{attribute 'linkalways'}
{attribute 'no_explicit_call' := 'This FB is a CLASS and must be accessed using methods or properties'}
{attribute 'enable_dynamic_creation'}
FUNCTION_BLOCK _ETcVnDetectBarcodesWalshOptions EXTENDS EnumDatatypeBase
VAR
	localData : ETcVnDetectBarcodesWalshOptions;
	activeData : REFERENCE TO ETcVnDetectBarcodesWalshOptions;
	enumBaseDatatype : _UDINT(localData);
END_VAR

METHOD PRIVATE AddLocalEnumeration
VAR_INPUT
	Enumeration : T_MAXSTRING;
	Value : ETcVnDetectBarcodesWalshOptions;
END_VAR
AddEnumeration(Enumeration, Value);
END_METHOD

PROPERTY PUBLIC Address : PVOID
GET
Address := ADR(activeData);
END_GET
END_PROPERTY

METHOD PUBLIC ClearReference
VAR_INPUT
END_VAR
activeData REF= localData;
SetBaseDatatypeReference();
END_METHOD

METHOD PUBLIC Clone : I_Datatype
VAR
    pClone : POINTER TO _ETcVnDetectBarcodesWalshOptions;
END_VAR
pClone := __NEW(_ETcVnDetectBarcodesWalshOptions(InitialValue := Value));
IF pClone = 0 THEN
    RETURN;
END_IF
Clone := pClone^;
END_METHOD

METHOD FB_init : BOOL
VAR_INPUT
	bInitRetains : BOOL; // if TRUE, the retain variables are initialized (warm start / cold start)
	bInCopyCode : BOOL;  // if TRUE, the instance afterwards gets moved into the copy code (online change)
	InitialValue : ETcVnDetectBarcodesWalshOptions;
END_VAR
localData := InitialValue;
AddBaseDatatype(enumBaseDatatype);
ClearReference();

AddLocalEnumeration('TCVN_DBWO_HORIZONTAL', ETcVnDetectBarcodesWalshOptions.TCVN_DBWO_HORIZONTAL);
AddLocalEnumeration('TCVN_DBWO_VERTICAL', ETcVnDetectBarcodesWalshOptions.TCVN_DBWO_VERTICAL);
AddLocalEnumeration('TCVN_DBWO_DIAGONAL_45', ETcVnDetectBarcodesWalshOptions.TCVN_DBWO_DIAGONAL_45);
AddLocalEnumeration('TCVN_DBWO_DIAGONAL_135', ETcVnDetectBarcodesWalshOptions.TCVN_DBWO_DIAGONAL_135);
AddLocalEnumeration('TCVN_DBWO_ALL_DIRECTIONS', ETcVnDetectBarcodesWalshOptions.TCVN_DBWO_ALL_DIRECTIONS);
END_METHOD

PROPERTY PUBLIC Identifier : T_MAXSTRING
GET
Identifier := 'ETcVnDetectBarcodesWalshOptions';
END_GET
END_PROPERTY

METHOD IsEnumeratorValueEqual : BOOL
VAR_INPUT
	Enumerator : I_KeyValueForwardEnumerator;
END_VAR
VAR
	storedValue : ETcVnDetectBarcodesWalshOptions;
END_VAR
IF NOT Enumerator.TryGet(storedValue) THEN
	RETURN;
END_IF

IsEnumeratorValueEqual := storedValue = activeData;
END_METHOD

METHOD PUBLIC MakeReferenceTo
VAR_INPUT
	ReferenceTarget : REFERENCE TO ETcVnDetectBarcodesWalshOptions;
END_VAR
activeData REF= ReferenceTarget;
SetBaseDatatypeReference();
END_METHOD

METHOD PROTECTED SetBaseDatatypeReference
VAR_INPUT
END_VAR
enumBaseDatatype.MakeReferenceTo(activeData);
END_METHOD

PROPERTY PUBLIC Size : UDINT
GET
Size := SIZEOF(activeData);
END_GET
END_PROPERTY

METHOD TryMakeReferenceTo : BOOL
VAR_INPUT
	Target : I_Datatype;
END_VAR
VAR
	pTargetData : POINTER TO ETcVnDetectBarcodesWalshOptions;
END_VAR
IF NOT IsEquivalentTo(Target) THEN
	RETURN;
END_IF

pTargetData := Target.Address;
activeData REF= pTargetData^;
SetBaseDatatypeReference();
TryMakeReferenceTo := TRUE;
END_METHOD

PROPERTY PUBLIC Value : ETcVnDetectBarcodesWalshOptions
GET
Value := activeData;
END_GET
SET
activeData := Value;
END_SET
END_PROPERTY

END_FUNCTION_BLOCK

(* stored: Version 1.1.0.1, ProductVersion 3.1.4026.13
   POU _ETcVnDetectBarcodesWalshOptions: Id {05084adb-6e52-4f98-af76-1434c289e7bb}, SpecialFunc None
   Folder Core: Id {d6fe9b04-bab6-4b89-a856-fce334837956}
   Folder Protected: Id {ce713da5-b68f-48a7-b3d8-2b84537450eb}
   Folder Customize: Id {b3346b1e-ca4f-4179-ac20-139bdbb97d4f}
   Folder Constructor: Id {8c1409ab-314d-4d9f-a2b6-4a18ce1050a5}
   Folder Private: Id {5ed77874-2200-4fc7-aa15-ad640a08b651}
   Folder Protected: Id {979a1b2c-7faf-42fc-adfb-7722c6e58b36}
   Method AddLocalEnumeration: Id {f0d147f6-a17e-4d64-b46d-004b88a218c0}
   Property Address: Id {7d0c229c-170c-4c53-b3df-e9d438e36930}
   Get Get: Id {0bc2dce1-3ba7-4e25-bc84-8522325ef36a}
   Method ClearReference: Id {7f4986f0-1bb0-45c4-9f05-f83a87e983bd}
   Method Clone: Id {487a9c2d-8c86-4ec0-8d54-42f749f680dd}
   Method FB_init: Id {b39ec7df-b847-4e29-a1df-84bd5a9254c1}
   Property Identifier: Id {57709980-79ca-474f-8767-0cf4dfffd9eb}
   Get Get: Id {ce3b2027-611b-4f92-95e6-cea4faf77425}
   Method IsEnumeratorValueEqual: Id {baf9f37e-9a41-4d84-a1fd-fce9b6d7824d}
   Method MakeReferenceTo: Id {46b22653-ab7e-4db8-9703-864475ad3a35}
   Method SetBaseDatatypeReference: Id {6c0bf3a4-3703-420b-929a-5e7420894c86}
   Property Size: Id {e5a9dba3-8945-4731-935b-9a61104efd44}
   Get Get: Id {3587f60b-735b-4b0f-a38d-3048ff1338bc}
   Method TryMakeReferenceTo: Id {0f5a7eb3-f532-456f-a7e3-b577f2eca924}
   Property Value: Id {566113cd-288b-49b3-9093-bdc516cba1f1}
   Get Get: Id {99afee35-f8b3-41ad-8ba5-55825f95c301}
   Set Set: Id {615894f2-a554-467d-bf4f-4cbb984ff6a6} *)
